Universal Robots PolyScope program: letter c.urp

Program letter c (installation=default directory=/programs/usbdisk createdIn=5.10.2.106319 lastSavedIn=5.10.2.106319 robotSerialNumber=20195501559)
Calibrated DH parameters: a=[0.000047, -0.411824, -0.383036, 0.00008, -0.000001, 0]; d=[0.162664, 43.611781, -55.695621, 12.217376, 0.099809, 0.099502]; alpha=[1.569652, -0.002418, 0.007042, 1.570603, -1.569925, 0]; deltaTheta=[0, -0.250699, 6.315302, 0.218595, 0.000001, 0]
Robot Program (runOnlyOnce=false)
  MoveP speed 250 mm/s, acceleration 1200 mm/s^2 (blendRadius=0.018 useActiveTCP=true) feature=Base
    Waypoint Waypoint_1: motionParameters(blendRadius=0.018); TCP in base x=-812.547 y=-185.02 z=98.967 mm, rx=2.5651 ry=1.8138 rz=0 rad; joints [3.535, -29.378, 55.383, -115.956, -89.772, 23.208] deg
    CircleMove (OrientationMode=UNCONSTRAINED)
      Waypoint ViaPoint_1: motionParameters(blendRadius=0.017); TCP in base x=-786.396 y=-158.18 z=97.885 mm, rx=-2.5649 ry=-1.8135 rz=0.0007 rad; joints [1.708, -33.632, 64.291, -120.639, -89.776, 21.424] deg
      Waypoint Waypoint_1: TCP in base x=-812.547 y=-185.02 z=98.967 mm, rx=2.5651 ry=1.8138 rz=0 rad; joints [3.535, -29.378, 55.383, -115.956, -89.772, 23.208] deg
  MoveP speed 250 mm/s, acceleration 1200 mm/s^2 (blendRadius=0.019 useActiveTCP=true) feature=Base
    Waypoint Waypoint_1: motionParameters(blendRadius=0.018); TCP in base x=-812.547 y=-185.02 z=98.967 mm, rx=2.5651 ry=1.8138 rz=0 rad; joints [3.535, -29.378, 55.383, -115.956, -89.772, 23.208] deg
    CircleMove (OrientationMode=UNCONSTRAINED)
      Waypoint ViaPoint_1: TCP in base x=-786.396 y=-158.18 z=97.885 mm, rx=-2.5649 ry=-1.8135 rz=0.0007 rad; joints [1.708, -33.632, 64.291, -120.639, -89.776, 21.424] deg
      Waypoint Waypoint_1: TCP in base x=-812.547 y=-185.02 z=98.967 mm, rx=2.5651 ry=1.8138 rz=0 rad; joints [3.535, -29.378, 55.383, -115.956, -89.772, 23.208] deg
  MoveJ speed 60 deg/s, acceleration 80 deg/s^2 (useActiveTCP=true) feature=Base
    Waypoint Waypoint_1: TCP in base x=-812.547 y=-185.02 z=98.967 mm, rx=2.5651 ry=1.8138 rz=0 rad; joints [3.535, -29.378, 55.383, -115.956, -89.772, 23.208] deg
